# EPICS autosave request: iocBoot/ioc13Mjolnir/auto_settings.req
file "E1608_settings.req",  P=$(E1608_PREFIX)
file "ISCO_settings.req",   P=$(ISCO_PREFIX)
file "Vindum_settings.req", P=$(VINDUM_PREFIX)
